// TIA Portal V18 export
DATA_BLOCK "Data_block_1"   // DB1
{ S7_Optimized_Access := 'TRUE' }
VERSION : 0.1
// stored: AutoNumber true, IsOnlyStoredInLoadMemory false, IsRetainMemResEnabled false, IsWriteProtectedInAS false, MemoryReserve 100
   VAR
      tag_1 : Real;
      tag_2 : Real;
      tag_3 : Real;
      tag_4 : Real;
      tag_5 : Real;
      tag_6 : Real;
      tag_7 : Real;
      tag_8 : Real;
      tag_9 : Real;
      tag_10 : Real;
      tag_11 : Real;
      tag_12 : Real;
      tag_13 : Real;
   END_VAR
BEGIN
END_DATA_BLOCK
